(* PLC project Sem nome, Desconhecido Sem nome 1 *)
(* stored: creationDateTime 2023-12-06T19:26:37, modificationDateTime 2025-02-10T17:12:32 *)

PROGRAM AWS
  VAR
    SP AT %QW0 : UINT;  (* SetPoint *)
    PV AT %IW0 : UINT;  (* Sinal Entrada *)
    CV AT %QW1 : UINT;  (* Sinal Controle *)
    ITERM AT %QD1 : REAL;
    error AT %QD2 : REAL;  (* Erro do sistema *)
    KP AT %QW2 : UINT;  (* Contante Proporcional *)
    KI AT %QW3 : UINT;  (* Ganho Integral *)
    R1 AT %IW4 : BOOL;  (* Reset bloco integração *)
  END_VAR
  VAR
    INTEGRAL0 : INTEGRAL;
  END_VAR

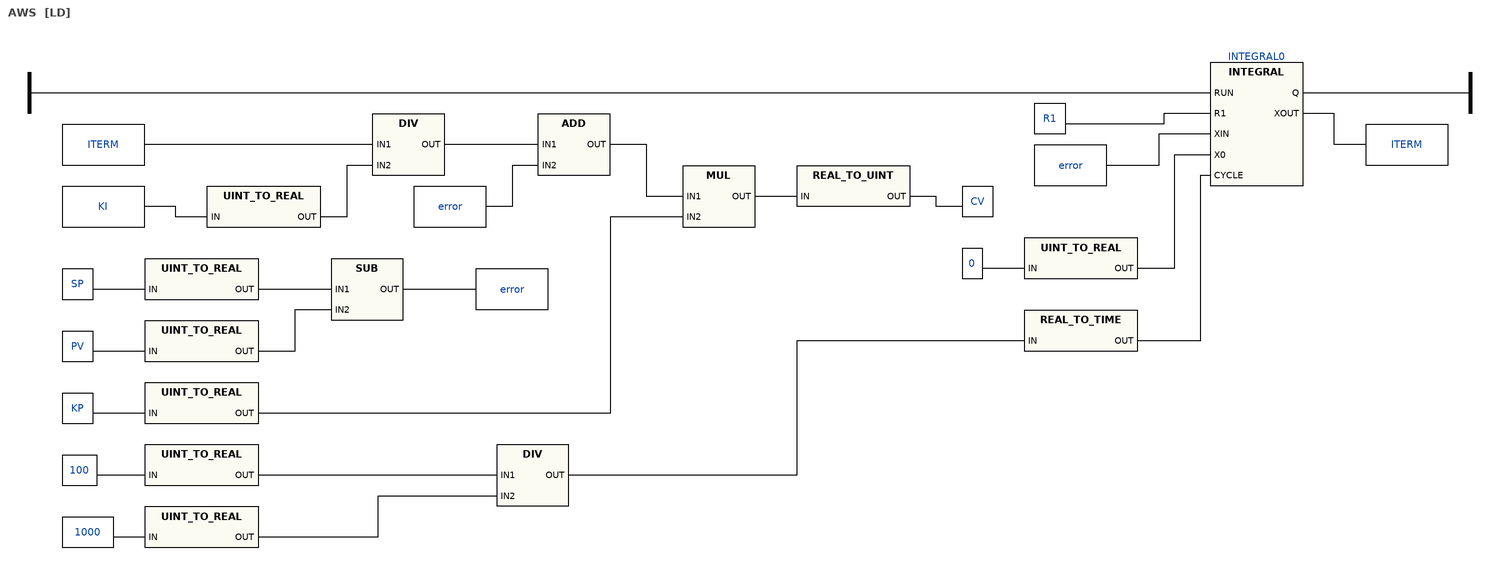
(* LD diagram, written out as Structured Text *)
CV := REAL_TO_UINT((ITERM / UINT_TO_REAL(KI) + error) * UINT_TO_REAL(KP));
error := UINT_TO_REAL(SP) - UINT_TO_REAL(PV);
INTEGRAL0(RUN := TRUE, R1 := R1, XIN := error, X0 := UINT_TO_REAL(0), CYCLE := REAL_TO_TIME(UINT_TO_REAL(100) / UINT_TO_REAL(1000)));
ITERM := INTEGRAL0.XOUT;
END_PROGRAM

CONFIGURATION Config0
  RESOURCE Res0 ON PLC
    TASK task0(INTERVAL := T#20ms, PRIORITY := 0);
    PROGRAM instance0 WITH task0 : AWS;
  END_RESOURCE
END_CONFIGURATION
